// TIA Portal V20 export
DATA_BLOCK "ErrTextList"   // DB371
{ S7_Optimized_Access := 'TRUE' }
// stored: AutoNumber false, MemoryReserve 0
   VAR RETAIN
      language : Array[1..10] of WString[2];   // language for alarm text [ISO639-1]
   END_VAR
   VAR
      writeMessage : Bool;   // write message from program to data block
      err : Array[2000..2205] of Struct   // alarm text
         idProd : UInt;   // producer Id (for Plc: 0=Program_Alarm, 4=SysDiag, 5=MotionControl, 6=Security, 8=GRAPH, 9=ProDiag)
         id : UInt;   // alarm Id
         prio : UInt;   // 0 .. 16 (0-1=info, 2=safety, 3=warning, 4-16=fault)
         alarm : Array[1..8] of WString[150];   // alarm text
      END_STRUCT;
   END_VAR
BEGIN
   language[1] := WSTRING#'de';
   language[2] := WSTRING#'en';
   language[3] := WSTRING#'it';
   language[4] := WSTRING#'fr';
   language[5] := WSTRING#'es';
   err[2031..2040].idProd := 0;
   err[2160..2167].idProd := 0;
   err[2170..2177].idProd := 0;
   err[2180..2187].idProd := 0;
   err[2031..2040].id := 0;
   err[2160..2167].id := 0;
   err[2170..2177].id := 0;
   err[2180..2187].id := 0;
   err[2000..2002].prio := 2;
   err[2004..2005].prio := 2;
   err[2010..2011].prio := 2;
   err[2013..2014].prio := 2;
   err[2016..2017].prio := 2;
   err[2019..2020].prio := 2;
   err[2030..2031].prio := 2;
   err[2032].prio := 0;
   err[2033..2040].prio := 2;
   err[2050].prio := 1;
   err[2052].prio := 0;
   err[2054].prio := 1;
   err[2060].prio := 10;
   err[2075].prio := 2;
   err[2080..2083].prio := 11;
   err[2090..2091].prio := 9;
   err[2100..2102].prio := 10;
   err[2110].prio := 8;
   err[2111].prio := 0;
   err[2120].prio := 12;
   err[2121..2125].prio := 7;
   err[2150].prio := 11;
   err[2151].prio := 10;
   err[2152..2153].prio := 8;
   err[2154].prio := 1;
   err[2156].prio := 1;
   err[2160].prio := 11;
   err[2161].prio := 10;
   err[2162..2163].prio := 8;
   err[2164].prio := 1;
   err[2165].prio := 0;
   err[2166].prio := 1;
   err[2167].prio := 0;
   err[2170].prio := 11;
   err[2171].prio := 10;
   err[2172..2173].prio := 8;
   err[2174].prio := 1;
   err[2175].prio := 0;
   err[2176].prio := 1;
   err[2177].prio := 0;
   err[2180].prio := 11;
   err[2181].prio := 10;
   err[2182..2183].prio := 8;
   err[2184].prio := 1;
   err[2185].prio := 0;
   err[2186].prio := 1;
   err[2187].prio := 0;
   err[2189].prio := 8;
   err[2190].prio := 9;
   err[2000].alarm[1] := WSTRING#'PLC - Not Aus Taster gedrückt am Pc Terminal (-14SB0+HMI.GLD)';
   err[2000].alarm[2] := WSTRING#'PLC - Emergency stop pressed at Pc terminal (-14SB0+HMI.GLD)';
   err[2000].alarm[3] := WSTRING#'PLC - Tasto per arresto di emergenza premuto sul terminale Pc (-14SB0+HMI.GLD)';
   err[2000].alarm[4] := WSTRING#'PLC - Arrêt d`urgence appuyé sur le terminal PC (-14SB0+HMI.GLD)';
   err[2000].alarm[5] := WSTRING#'PLC - Parada de emergencia presionada en terminal Pc (-14SB0+HMI.GLD)';
   err[2001].alarm[1] := WSTRING#'PLC - Not Aus Schlüsselschalter ausgeschalten am Pc Terminal (-14SB1+HMI.GLD)';
   err[2001].alarm[2] := WSTRING#'PLC - Emergency enable key switch off at Pc terminal (-14SB1+HMI.GLD)';
   err[2001].alarm[3] := WSTRING#'PLC - Interruttore a chiave per aresto di emergenza spento sul terminale del PC (-14SB1+HMI.GLD)';
   err[2001].alarm[4] := WSTRING#'PLC - Interrupteur d`urgence désactivé sur le terminal PC (-14SB1+HMI.GLD)';
   err[2001].alarm[5] := WSTRING#'PLC - Interruptor de llave de parada de emergencia apagado en la terminal de la PC (-14SB1+HMI.GLD)';
   err[2002].alarm[1] := WSTRING#'PLC - Quittierung notwendig für Not Aus Taster/Schlüsselschalter am Pc Terminal (-14SB0/1+HMI.GLD)';
   err[2002].alarm[2] := WSTRING#'PLC - Acknowledge required for emergency stop/key switch at Pc terminal (-14SB0/1+HMI.GLD)';
   err[2002].alarm[3] := WSTRING#'PLC - Reset richiesto per pulsante/interrutore di arresto di emergenza sul terminale PC (-14SB0/1+HMI.GLD)';
   err[2002].alarm[4] := WSTRING#'PLC - Reconnaissance nécessaire pour l`arrêt d`urgence/interrupteur à clé sur le terminal PC (-14SB0/1+HMI.GLD)';
   err[2002].alarm[5] := WSTRING#'PLC - Es necesario reiniciar para el botónIinterruptor de emergencia en terminal de PC (-14SB0/1+HMI.GLD)';
   err[2004].alarm[1] := WSTRING#'PLC - Not Aus von externe machine (-XNA+SGV) - aktiv';
   err[2004].alarm[2] := WSTRING#'PLC - Emergency stop from external machine (-XNA+SGV) - active';
   err[2004].alarm[3] := WSTRING#'PLC - Arresto di emergenza da macchina esterna (-XNA+SGV) - attivo';
   err[2004].alarm[4] := WSTRING#'PLC - Arrêt d`urgence depuis une machine externe (-XNA+SGV) - actif';
   err[2004].alarm[5] := WSTRING#'PLC - Parada de emergencia desde máquina externa (-XNA+SGV) - activo';
   err[2005].alarm[1] := WSTRING#'PLC - Not Aus von externe machine (-XNA+SGV) - Quittierung notwendig';
   err[2005].alarm[2] := WSTRING#'PLC - Emergency stop from external machine (-XNA+SGV) - acknowledgement required';
   err[2005].alarm[3] := WSTRING#'PLC - Arresto di emergenza da macchina esterna (-XNA+SGV) - reset necessario';
   err[2005].alarm[4] := WSTRING#'PLC - Arrêt d`urgence depuis une machine externe (-XNA+SGV) - réinitialiser requis';
   err[2005].alarm[5] := WSTRING#'PLC - Parada de emergencia desde máquina externa (-XNA+SGV) - es necesario reiniciar';
   err[2010].alarm[1] := WSTRING#'PLC - Sicherheitsschalter -14SS1.TL+SGV bei Scanner für visuelle Beurteilung oben links - open';
   err[2010].alarm[2] := WSTRING#'PLC - Safety switch -14SS1.TL+SGV at scanner for visual measurement top left - open';
   err[2010].alarm[3] := WSTRING#'PLC - Interruttore di sicurezza -14SS1.TL+SGV sullo scanner per misurazione visiva in alto a sinistra - aperto';
   err[2010].alarm[4] := WSTRING#'PLC - interrupteur de sécurité -14SS1.TL+SGV au scanner pour mesure visuelle en haut à gauche - ouvert';
   err[2010].alarm[5] := WSTRING#'PLC - interruptor de seguridad -14SS1.TL+SGV en el escáner para medición visual arriba a la izquierda - abierto';
   err[2011].alarm[1] := WSTRING#'PLC - Sicherheitsschalter -14SS1.TL+SGV bei Scanner für visuelle Beurteilung oben links - Quittierung notwendig';
   err[2011].alarm[2] := WSTRING#'PLC - safety switch -14SS1.TL+SGV at scanner for visual measurement top left - acknowledge required';
   err[2011].alarm[3] := WSTRING#'PLC - Interruttore di sicurezza -14SS1.TL+SGV sullo scanner per misurazione visiva in alto a sinistra - reset necessario';
   err[2011].alarm[4] := WSTRING#'PLC - interrupteur de sécurité -14SS1.TL+SGV au scanner pour mesure visuelle en haut à gauche - réinitialiser requis';
   err[2011].alarm[5] := WSTRING#'PLC - interruptor de seguridad -14SS1.TL+SGV en el escáner para medición visual arriba a la izquierda - es necesario reiniciar';
   err[2013].alarm[1] := WSTRING#'PLC - Sicherheitsschalter -14SS1.BL+SGV bei Scanner für visuelle Beurteilung unten links - open';
   err[2013].alarm[2] := WSTRING#'PLC - Safety switch -14SS1.BL+SGV at scanner for visual measurement bottom left - open';
   err[2013].alarm[3] := WSTRING#'PLC - Interruttore di sicurezza -14SS1.BL+SGV sullo scanner per misurazione visiva in basso a sinistra - aperto';
   err[2013].alarm[4] := WSTRING#'PLC - interrupteur de sécurité -14SS1.BL+SGV au scanner pour mesure visuelle en bas à gauche - ouvert';
   err[2013].alarm[5] := WSTRING#'PLC - interruptor de seguridad -14SS1.BL+SGV en el escáner para medición visual abajoa la izquierda - abierto';
   err[2014].alarm[1] := WSTRING#'PLC - Sicherheitsschalter -14SS1.BL+SGV bei Scanner für visuelle Beurteilung unten links - Quittierung notwendig';
   err[2014].alarm[2] := WSTRING#'PLC - Safety switch -14SS1.BL+SGV at scanner for visual measurement bottom left - acknowledge required';
   err[2014].alarm[3] := WSTRING#'PLC - Interruttore di sicurezza -14SS1.BL+SGV sullo scanner per misurazione visiva in basso a sinistra - reset necessario';
   err[2014].alarm[4] := WSTRING#'PLC - interrupteur de sécurité -14SS1.BL+SGV au scanner pour mesure visuelle en bas à gauche - réinitialiser requis';
   err[2014].alarm[5] := WSTRING#'PLC - interruptor de seguridad -14SS1.BL+SGV en el escáner para medición visual abajoa la izquierda - es necesario reiniciar';
   err[2016].alarm[1] := WSTRING#'PLC - Sicherheitsschalter -14SS1.TR+SGV bei Scanner für visuelle Beurteilung oben rechts- open';
   err[2016].alarm[2] := WSTRING#'PLC - Safety switch -14SS1.TR+SGV at scanner for visual measurement top right - open';
   err[2016].alarm[3] := WSTRING#'PLC - Interruttore di sicurezza -14SS1.TR+SGV sullo scanner per misurazione visiva in alto a destra - aperto';
   err[2016].alarm[4] := WSTRING#'PLC - interrupteur de sécurité -14SS1.TR+SGV au scanner pour mesure visuelle en haut à droite - ouvert';
   err[2016].alarm[5] := WSTRING#'PLC - interruptor de seguridad -14SS1.TR+SGV en el escáner para medición visual arriba a la derecha - abierto';
   err[2017].alarm[1] := WSTRING#'PLC - Sicherheitsschalter -14SS1.TR+SGV bei Scanner für visuelle Beurteilung oben rechts- Quittierung notwendig';
   err[2017].alarm[2] := WSTRING#'PLC - Safety switch -14SS1.TR+SGV at scanner for visual measurement top right -  acknowledge required';
   err[2017].alarm[3] := WSTRING#'PLC - Interruttore di sicurezza -14SS1.TR+SGV sullo scanner per misurazione visiva in alto a destra - reset necessario';
   err[2017].alarm[4] := WSTRING#'PLC - interrupteur de sécurité -14SS1.TR+SGV au scanner pour mesure visuelle en haut à droite - réinitialiser requis';
   err[2017].alarm[5] := WSTRING#'PLC - interruptor de seguridad -14SS1.TR+SGV en el escáner para medición visual arriba a la derecha - es necesario reiniciar';
   err[2019].alarm[1] := WSTRING#'PLC - Sicherheitsschalter -14SS1.BR+SGV bei Scanner für visuelle Beurteilung unten rechts - open';
   err[2019].alarm[2] := WSTRING#'PLC - Safety switch -14SS1.BR+SGV at scanner for visual measurement bottom right - open';
   err[2019].alarm[3] := WSTRING#'PLC - Interruttore di sicurezza -14SS1.BR+SGV sullo scanner per misurazione visiva in basso a destra - aperto';
   err[2019].alarm[4] := WSTRING#'PLC - interrupteur de sécurité -14SS1.BR+SGV au scanner pour mesure visuelle en bas à droite - ouvert';
   err[2019].alarm[5] := WSTRING#'PLC - interruptor de seguridad -14SS1.BR+SGV en el escáner para medición visual abajo a la derecha - abierto';
   err[2020].alarm[1] := WSTRING#'PLC - Sicherheitsschalter -14SS1.BR+SGV bei Scanner für visuelle Beurteilung unten rechts - Quittierung notwendig';
   err[2020].alarm[2] := WSTRING#'PLC - Safety switch -14SS1.BR+SGV at scanner for visual measurement bottom right -  acknowledge required';
   err[2020].alarm[3] := WSTRING#'PLC - Interruttore di sicurezza -14SS1.BR+SGV sullo scanner per misurazione visiva in basso a destra - reset necessario';
   err[2020].alarm[4] := WSTRING#'PLC - interrupteur de sécurité -14SS1.BR+SGV au scanner pour mesure visuelle en bas à droite - réinitialiser requis';
   err[2020].alarm[5] := WSTRING#'PLC - interruptor de seguridad -14SS1.BR+SGV en el escáner para medición visual abajo a la derecha - es necesario reiniciar';
   err[2030].alarm[1] := WSTRING#'PLC - Sicherheitsschalter -14SS1.TL+SGX bei Scanner für X-Ray oben links - open';
   err[2030].alarm[2] := WSTRING#'PLC - Safety switch -14SS1.TL+SGX at scanner for X-Ray top left - open';
   err[2030].alarm[3] := WSTRING#'PLC - Interruttore di sicurezza -14SS1.TL+SGX sullo scanner per X-Ray in alto a sinistra - aperto';
   err[2030].alarm[4] := WSTRING#'PLC - interrupteur de sécurité -14SS1.TL+SGX au scanner pour X-Ray en haut à gauche - ouvert';
   err[2030].alarm[5] := WSTRING#'PLC - interruptor de seguridad -14SS1.TL+SGX en el escáner para X-Ray arriba a la izquierda - abierto';
   err[2030].alarm[6..8] := WSTRING#'';
   err[2031].alarm[1] := WSTRING#'PLC - Sicherheitsschalter -14SS1.TL+SGX bei Scanner für X-Ray oben links - Quittierung notwendig';
   err[2031].alarm[2] := WSTRING#'PLC - safety switch -14SS1.TL+SGX at scanner for X-Ray top left - acknowledge required';
   err[2031].alarm[3] := WSTRING#'PLC - Interruttore di sicurezza -14SS1.TL+SGX sullo scanner per X-Ray in alto a sinistra - reset necessario';
   err[2031].alarm[4] := WSTRING#'PLC - interrupteur de sécurité -14SS1.TL+SGX au scanner pour X-Ray en haut à gauche - réinitialiser requis';
   err[2031].alarm[5] := WSTRING#'PLC - interruptor de seguridad -14SS1.TL+SGX en el escáner para X-Ray arriba a la izquierda - es necesario reiniciar';
   err[2031].alarm[6..8] := WSTRING#'';
   err[2032].alarm[1..8] := WSTRING#'';
   err[2033].alarm[1] := WSTRING#'PLC - Sicherheitsschalter -14SS1.BL+SGX bei Scanner für X-Ray unten links - open';
   err[2033].alarm[2] := WSTRING#'PLC - Safety switch -14SS1.BL+SGX at scanner for X-Ray bottom left - open';
   err[2033].alarm[3] := WSTRING#'PLC - Interruttore di sicurezza -14SS1.BL+SGX sullo scanner per X-Ray in basso a sinistra - aperto';
   err[2033].alarm[4] := WSTRING#'PLC - interrupteur de sécurité -14SS1.BL+SGX au scanner pour X-Ray en bas à gauche - ouvert';
   err[2033].alarm[5] := WSTRING#'PLC - interruptor de seguridad -14SS1.BL+SGX en el escáner para X-Ray abajoa la izquierda - abierto';
   err[2033].alarm[6..8] := WSTRING#'';
   err[2034].alarm[1] := WSTRING#'PLC - Sicherheitsschalter -14SS1.BL+SGX bei Scanner für X-Ray unten links - Quittierung notwendig';
   err[2034].alarm[2] := WSTRING#'PLC - Safety switch -14SS1.BL+SGX at scanner for X-Rayt bottom left - acknowledge required';
   err[2034].alarm[3] := WSTRING#'PLC - Interruttore di sicurezza -14SS1.BL+SGX sullo scanner per X-Ray in basso a sinistra - reset necessario';
   err[2034].alarm[4] := WSTRING#'PLC - interrupteur de sécurité -14SS1.BL+SGX au scanner pour X-Ray en bas à gauche - réinitialiser requis';
   err[2034].alarm[5] := WSTRING#'PLC - interruptor de seguridad -14SS1.BL+SGX en el escáner para X-Ray abajoa la izquierda - es necesario reiniciar';
   err[2034].alarm[6..8] := WSTRING#'';
   err[2035].alarm[1..8] := WSTRING#'';
   err[2036].alarm[1] := WSTRING#'PLC - Sicherheitsschalter -14SS1.TR+SGX bei Scanner für X-Ray oben rechts- open';
   err[2036].alarm[2] := WSTRING#'PLC - Safety switch -14SS1.TR+SGX at scanner for X-Ray top right - open';
   err[2036].alarm[3] := WSTRING#'PLC - Interruttore di sicurezza -14SS1.TR+SGX sullo scanner per X-Ray in alto a destra - aperto';
   err[2036].alarm[4] := WSTRING#'PLC - interrupteur de sécurité -14SS1.TR+SGX au scanner pour X-Ray en haut à droite - ouvert';
   err[2036].alarm[5] := WSTRING#'PLC - interruptor de seguridad -14SS1.TR+SGX en el escáner para X-Ray arriba a la derecha - abierto';
   err[2036].alarm[6..8] := WSTRING#'';
   err[2037].alarm[1] := WSTRING#'PLC - Sicherheitsschalter -14SS1.TR+SGX bei Scanner für X-Ray oben rechts- Quittierung notwendig';
   err[2037].alarm[2] := WSTRING#'PLC - Safety switch -14SS1.TR+SGX at scanner for X-Ray top right -  acknowledge required';
   err[2037].alarm[3] := WSTRING#'PLC - Interruttore di sicurezza -14SS1.TR+SGX sullo scanner per X-Ray in alto a destra - reset necessario';
   err[2037].alarm[4] := WSTRING#'PLC - interrupteur de sécurité -14SS1.TR+SGX au scanner pour X-Ray en haut à droite - réinitialiser requis';
   err[2037].alarm[5] := WSTRING#'PLC - interruptor de seguridad -14SS1.TR+SGX en el escáner para X-Ray arriba a la derecha - es necesario reiniciar';
   err[2037].alarm[6..8] := WSTRING#'';
   err[2038].alarm[1..8] := WSTRING#'';
   err[2039].alarm[1] := WSTRING#'PLC - Sicherheitsschalter -14SS1.BR+SGX bei Scanner für X-Ray unten rechts - open';
   err[2039].alarm[2] := WSTRING#'PLC - Safety switch -14SS1.BR+SGX at scanner for X-Ray bottom right - open';
   err[2039].alarm[3] := WSTRING#'PLC - Interruttore di sicurezza -14SS1.BR+SGX sullo scanner per X-Ray in basso a destra - aperto';
   err[2039].alarm[4] := WSTRING#'PLC - interrupteur de sécurité -14SS1.BR+SGX au scanner pour X-Ray en bas à droite - ouvert';
   err[2039].alarm[5] := WSTRING#'PLC - interruptor de seguridad -14SS1.BR+SGX en el escáner para X-Ray abajo a la derecha - abierto';
   err[2039].alarm[6..8] := WSTRING#'';
   err[2040].alarm[1] := WSTRING#'PLC - Sicherheitsschalter -14SS1.BR+SGX bei Scanner für X-Ray unten rechts - Quittierung notwendig';
   err[2040].alarm[2] := WSTRING#'PLC - Safety switch -14SS1.BR+SGX at scanner for X-Ray bottom right -  acknowledge required';
   err[2040].alarm[3] := WSTRING#'PLC - Interruttore di sicurezza -14SS1.BR+SGX sullo scanner per X-Ray in basso a destra - reset necessario';
   err[2040].alarm[4] := WSTRING#'PLC - interrupteur de sécurité -14SS1.BR+SGX au scanner pour X-Ray en bas à droite - réinitialiser requis';
   err[2040].alarm[5] := WSTRING#'PLC - interruptor de seguridad -14SS1.BR+SGX en el escáner para X-Ray abajo a la derecha - es necesario reiniciar';
   err[2050].alarm[1] := WSTRING#'PLC - Schlüsselschalter für Einrichtbetrieb am Scanner links aktiviert (-14SB1+SSTL)';
   err[2050].alarm[2] := WSTRING#'PLC - setting mode key switch at scanner left active (-14SB1+SSTL)';
   err[2050].alarm[3] := WSTRING#'PLC - Interruttore a chiave per la modalità di impostazione attivato sullo scanner a sinistra (-14SB1+SSTL)';
   err[2050].alarm[4] := WSTRING#'PLC - commutateur à clé du mode de réglage à gauche du scanner actif (-14SB1+SSTL)';
   err[2050].alarm[5] := WSTRING#'PLC - interruptor de modo de ajuste a la izquierda del escáner activo (-14SB1+SSTL)';
   err[2052].alarm[1] := WSTRING#'PLC - Taster für Freigabe Verstellungen am Scanner links aktiviert (-14SB2+SSTL)';
   err[2052].alarm[2] := WSTRING#'PLC - button to enable adjustments at scanner left active (-14SB21+SSTL)';
   err[2052].alarm[3] := WSTRING#'PLC - pulsante per abilitare le assi attivato sullo scanner a sinistra (-14SB2+SSTL)';
   err[2052].alarm[4] := WSTRING#'PLC - bouton pour activer les réglages à gauche du scanner actif (-14SB2+SSTL)';
   err[2052].alarm[5] := WSTRING#'PLC - botón para habilitar ajustes a la izquierda del escáner activo (-14SB2+SSTL)';
   err[2054].alarm[1] := WSTRING#'PLC - Kühlgeräte wurden am Scanner rechts deaktiviert (-14SB2+SSTL)';
   err[2054].alarm[2] := WSTRING#'PLC - air-conditioning is switched off at scanner right (-0SH1+SSTR)';
   err[2054].alarm[3] := WSTRING#'PLC - l`aria condizionata è stata spenta sullo scanner a destra (-14SB2+SSTL)';
   err[2054].alarm[4] := WSTRING#'PLC - la climatisation est éteinte au niveau du scanner à droite (-14SB2+SSTL)';
   err[2054].alarm[5] := WSTRING#'PLC - El aire acondicionado está apagado en el escáner a la derecha (-14SB2+SSTL)';
   err[2060].alarm[1] := WSTRING#'PLC - Störung Sicherheitsmodule';
   err[2060].alarm[2] := WSTRING#'PLC - fault safety modules plc';
   err[2060].alarm[3] := WSTRING#'PLC - errore sui moduli di sicurezza';
   err[2060].alarm[4] := WSTRING#'PLC - modules de sécurité contre les défauts';
   err[2060].alarm[5] := WSTRING#'PLC - módulos de seguridad contra fallas';
   err[2075].alarm[1] := WSTRING#'PLC - Sicherheitsbereich Extern oder Intern ausgeschalten - Quittierung notwendig';
   err[2075].alarm[2] := WSTRING#'PLC - safety area internal/external switched off - acknowledge required';
   err[2075].alarm[3] := WSTRING#'PLC - area di sicurezza interna/esterna spenta- reset necessario';
   err[2075].alarm[4] := WSTRING#'PLC - zone de sécurité interne/externe désactivée - réinitialiser requis';
   err[2075].alarm[5] := WSTRING#'PLC - area de seguridad interna/externa apagada - es necesario reiniciar';
   err[2080].alarm[1] := WSTRING#'PLC - Störung Rückführung Sicherheitsbereich - Bereich laser (-14KA1+SGV)';
   err[2080].alarm[2] := WSTRING#'PLC - fault safety feedback monitoring - area laser (-14KA1+SGV)';
   err[2080].alarm[3] := WSTRING#'PLC - errore monitoraggio feedback di sicurezza - area laser (-14KA1+SGV)';
   err[2080].alarm[4] := WSTRING#'PLC - défaut surveillance de la sécurité - zone laser (-14KA1+SGV)';
   err[2080].alarm[5] := WSTRING#'PLC - fallo de monitoreo de retroalimentación de seguridad - área de láser (-14KA1+SGV)';
   err[2081].alarm[1] := WSTRING#'PLC - Störung Rückführung Sicherheitsbereich - Bereich Verstellung (-14KA2+SGV)';
   err[2081].alarm[2] := WSTRING#'PLC - fault safety feedback monitoring - area adjustment (-14KA2+SGV)';
   err[2081].alarm[3] := WSTRING#'PLC - errore monitoraggio feedback di sicurezza - area posizionamento (-14KA2+SGV)';
   err[2081].alarm[4] := WSTRING#'PLC - défaut surveillance de la sécurité - zone réglage (-14KA2+SGV)';
   err[2081].alarm[5] := WSTRING#'PLC - fallo de monitoreo de retroalimentación de seguridad - área de ajuste (-14KA2+SGV)';
   err[2082].alarm[1] := WSTRING#'PLC - Störung Rückführung Sicherheitsbereich - Bereich Verstellung LINMOT (8U1+SGV)';
   err[2082].alarm[2] := WSTRING#'PLC - fault safety feedback monitoring - area adjustment LINMOT (8U1+SGV)';
   err[2082].alarm[3] := WSTRING#'PLC - errore monitoraggio feedback di sicurezza - area posizionamento LINMOT (8U1+SGV)';
   err[2082].alarm[4] := WSTRING#'PLC - défaut surveillance de la sécurité - zone réglage LINMOT (8U1+SGV)';
   err[2082].alarm[5] := WSTRING#'PLC - fallo de monitoreo de retroalimentación de seguridad - área de ajuste LINMOT (8U1+SGV)';
   err[2083].alarm[1] := WSTRING#'PLC - Störung Rückführung Sicherheitsbereich - Bereich X-Ray (-5AX1+SGX)';
   err[2083].alarm[2] := WSTRING#'PLC - fault safety feedback monitoring - area X-Ray (-5AX1+SGX)';
   err[2083].alarm[3] := WSTRING#'PLC - errore monitoraggio feedback di sicurezza - area X-Ray (-5AX1+SGX)';
   err[2083].alarm[4] := WSTRING#'PLC - défaut surveillance de la sécurité - zone X-Ray (-5AX1+SGX)';
   err[2083].alarm[5] := WSTRING#'PLC - fallo de monitoreo de retroalimentación de seguridad - área X-Ray (-5AX1+SGX)';
   err[2090].alarm[1] := WSTRING#'PLC - Störung Lichtschranke im Scanner für visuelle Beurteilung (-1BTR2+SGV)';
   err[2090].alarm[2] := WSTRING#'PLC - fault light barrier in scanner for visual measurement (-1BTR2+SGV)';
   err[2090].alarm[3] := WSTRING#'PLC - errore sensore nel scanner per misurazione visiva (-1BTR2+SGV)';
   err[2090].alarm[4] := WSTRING#'PLC - défaut capteur dans le scanner pour la mesure visuelle (-1BTR2+SGV)';
   err[2090].alarm[5] := WSTRING#'PLC - fallo de sensor en escáner para medición visual (-1BTR2+SGV)';
   err[2091].alarm[1] := WSTRING#'PLC - Störung Lichtschranke vor Scanner für X-Ray (-1BTR2+SGX)';
   err[2091].alarm[2] := WSTRING#'PLC - fault light barrier before scanner for X-Ray (-1BTR2+SGX)';
   err[2091].alarm[3] := WSTRING#'PLC - errore sensore prime dello scanner per X-Ray (-1BTR2+SGX)';
   err[2091].alarm[4] := WSTRING#'PLC - défaut capteur avant le scanner pour X-Ray (-1BTR2+SGX)';
   err[2091].alarm[5] := WSTRING#'PLC - fallo de sensor antes escáner para X-Ray (-1BTR2+SGX)';
   err[2100].alarm[1] := WSTRING#'PLC - Störung Encoder vor Scanner (-1BCI1+GLD)';
   err[2100].alarm[2] := WSTRING#'PLC - fault encoder before scanner (-1BCI1+GLD)';
   err[2100].alarm[3] := WSTRING#'PLC - errore encoder davanti allo scanner (-1BCI1+GLD)';
   err[2100].alarm[4] := WSTRING#'PLC - défaut codeur avant le scanner (-1BCI1+GLD)';
   err[2100].alarm[5] := WSTRING#'PLC - fallo de codificador antes escáner (-1BCI1+GLD)';
   err[2101].alarm[1] := WSTRING#'PLC - Störung Encoder im Scanner (-1BCM1+GLD)';
   err[2101].alarm[2] := WSTRING#'PLC - fault encoder in scanner (-1BCM1+GLD)';
   err[2101].alarm[3] := WSTRING#'PLC - errore encoder nello scanner (-1BCM1+GLD)';
   err[2101].alarm[4] := WSTRING#'PLC - défaut codeur dans le scanner (-1BCM1+GLD)';
   err[2101].alarm[5] := WSTRING#'PLC - fallo de codificador en escáner (-1BCM1+GLD)';
   err[2102].alarm[1] := WSTRING#'PLC - Störung Encoder nach Scanner (-1BCO1+GLD)';
   err[2102].alarm[2] := WSTRING#'PLC - fault encoder after scanner (-1BCO1+GLD)';
   err[2102].alarm[3] := WSTRING#'PLC - errore encoder dopo lo scanner (-1BCO1+GLD)';
   err[2102].alarm[4] := WSTRING#'PLC - défaut codeur après le scanner (-1BCO1+GLD)';
   err[2102].alarm[5] := WSTRING#'PLC - fallo de codificador después del escáner (-1BCO1+GLD)';
   err[2110].alarm[1] := WSTRING#'PLC - Störung Kommunikation mit Goldeneye Pc';
   err[2110].alarm[2] := WSTRING#'PLC - fault communication with Goldeneye Pc';
   err[2110].alarm[3] := WSTRING#'PLC - errore comunicazione con Goldeneye Pc';
   err[2110].alarm[4] := WSTRING#'PLC - défaut communication avec Goldeneye Pc';
   err[2110].alarm[5] := WSTRING#'PLC - fallo comunicación con Goldeneye Pc';
   err[2111].alarm[1] := WSTRING#'PLC - Keine Freigabe vom Goldeneye Pc für den Einzug';
   err[2111].alarm[2] := WSTRING#'PLC - no release from Goldeneye Pc to infeed';
   err[2111].alarm[3] := WSTRING#'PLC - nessun permesso dal Goldeneye Pc per alimentazione ';
   err[2111].alarm[4] := WSTRING#'PLC - pas de sortie de Goldeneye PC pour infeed';
   err[2111].alarm[5] := WSTRING#'PLC - no hay liberación de Goldeneye Pc para la entrada';
   err[2120].alarm[1] := WSTRING#'PLC - Störung elektronischer Schutzschalter (-0F1.1+SGV)';
   err[2120].alarm[2] := WSTRING#'PLC - fault electronic circuit breaker (-0F1.1+SGV)';
   err[2120].alarm[3] := WSTRING#'PLC - errore interruttore elettronico (-0F1.1+SGV)';
   err[2120].alarm[4] := WSTRING#'PLC - défaut disjoncteur électronique (-0F1.1+SGV)';
   err[2120].alarm[5] := WSTRING#'PLC - fallo disyuntor electrónico (-0F1.1+SGV)';
   err[2121].alarm[1] := WSTRING#'PLC - Störung Kühlgerät 1 bei Scanner für visuelle Beurteilung (-0E1+SGV)';
   err[2121].alarm[2] := WSTRING#'PLC - fault air-conditioning unit 1 for scannerhousing visual measurement (-0E1+SGV)';
   err[2121].alarm[3] := WSTRING#'PLC - errore unità di raffreddamento 1 per scanner per misurazione visiva (-0E1+SGV)';
   err[2121].alarm[4] := WSTRING#'PLC - défaut unité de refroidissement 1 chez scanner pour mesure visuelle (-0E1+SGV)';
   err[2121].alarm[5] := WSTRING#'PLC - fallo unidad de refrigeración 1 para escáner para medición visual (-0E1+SGV)';
   err[2122].alarm[1] := WSTRING#'PLC - Störung Kühlgerät bei Scanner für X-Ray (-0E2+SGX)';
   err[2122].alarm[2] := WSTRING#'PLC - fault air-conditioning unit for scannerhousing  X-Ray (-0E2+SGX)';
   err[2122].alarm[3] := WSTRING#'PLC - errore unità di raffreddamento per scanner per X-Ray (-0E2+SGX)';
   err[2122].alarm[4] := WSTRING#'PLC - défaut unité de refroidissement chez scanner pour X-Ray (-0E2+SGX)';
   err[2122].alarm[5] := WSTRING#'PLC - fallo unidad de refrigeración para escáner para X-Ray (-0E2+SGX)';
   err[2123].alarm[1] := WSTRING#'PLC - Störung Kühlgerät 2 bei Scanner für visuelle Beurteilung (-0E1.1+SGV)';
   err[2123].alarm[2] := WSTRING#'PLC - fault air-conditioning unit 2 for scannerhousing visual measurement (-0E1.1+SGV)';
   err[2123].alarm[3] := WSTRING#'PLC - errore unità di raffreddamento 2 per scanner per misurazione visiva (-0E1.1+SGV)';
   err[2123].alarm[4] := WSTRING#'PLC - défaut unité de refroidissement 2 chez scanner pour mesure visuelle (-0E1.1+SGV)';
   err[2123].alarm[5] := WSTRING#'PLC - fallo unidad de refrigeración 2 para escáner para medición visual (-0E1.1+SGV)';
   err[2124].alarm[1] := WSTRING#'PLC - Störung Entfeuchter bei Scanner für (-0E1.2+SGV)';
   err[2124].alarm[2] := WSTRING#'PLC - fault dehumidifier for scannerhousing (-0E1.2+SGV)';
   err[2124].alarm[3] := WSTRING#'PLC - errore deumidificatore per scanner (-0E1.2+SGV)';
   err[2124].alarm[4] := WSTRING#'PLC - défaut déshumidificateur chez scanner (-0E1.2+SGV)';
   err[2124].alarm[5] := WSTRING#'PLC - fallo deshumidificador para escáner (-0E1.2+SGV)';
   err[2125].alarm[1] := WSTRING#'PLC - Störung Kommunikationsschnittstelle zwischen Pc und Sps ist unterschiedlich';
   err[2125].alarm[2] := WSTRING#'PLC - fault communication interface between Pc and Plc is different';
   err[2125].alarm[3] := WSTRING#'PLC - errore l`interfaccia di comunicazione tra Pc e Plc è diversa';
   err[2125].alarm[4] := WSTRING#'PLC - défaut l`interface de communication entre le PC et Plc est différente';
   err[2125].alarm[5] := WSTRING#'PLC - fallo La interfaz de comunicación entre PC y PLC es diferente';
   err[2140].alarm[1] := WSTRING#'PLC - Verstellung Scanner wurde temporär deaktiviert, kann nur mehr manuel verfahren werden (-8M1.B+SGV)';
   err[2140].alarm[2] := WSTRING#'PLC - adjustment scannerhousing is deactivated temporaly, you can move only manualy (-8M1.B+SGV)';
   err[2140].alarm[3] := WSTRING#'PLC - posizionamento scanner è temporaneamente disattivato, è possibile muoverlo solo manualmente (-8M1.B+SGV)';
   err[2140].alarm[4] := WSTRING#'PLC - positionnement de scanner est temporairement désactivé, vous ne pouvez le déplacer que manuellement (-8M1.B+SGV)';
   err[2140].alarm[5] := WSTRING#'PLC - el ajuste de del escáner se desactiva temporalmente, solo se puede mover manualmente (-8M1.B+SGV)';
   err[2141].alarm[1] := WSTRING#'PLC - Verstellung Messbalken oben wurde temporär deaktiviert, kann nur mehr manuel verfahren werden (-8M1.T+SGV)';
   err[2141].alarm[2] := WSTRING#'PLC - adjustment metering bar top is deactivated temporaly, you can move only manualy (-8M1.T+SGV)';
   err[2141].alarm[3] := WSTRING#'PLC - posizionamento barra di misura superiore è temporaneamente disattivato, è possibile muoverlo solo manualmente (-8M1.T+SGV)';
   err[2141].alarm[4] := WSTRING#'PLC - positionnement de barre de mesure supérieure est temporairement désactivé, vous ne pouvez le déplacer que manuellement (-8M1.T+SGV)';
   err[2141].alarm[5] := WSTRING#'PLC - el ajuste de barra de medición superior se desactiva temporalmente, solo se puede mover manualmente (-8M1.T+SGV)';
   err[2142].alarm[1] := WSTRING#'PLC - Verstellung Messbalken links wurde temporär deaktiviert, kann nur mehr manuel verfahren werden (-8M1.L+SGV)';
   err[2142].alarm[2] := WSTRING#'PLC - adjustment metering bar left is deactivated temporaly, you can move only manualy (-8M1.L+SGV)';
   err[2142].alarm[3] := WSTRING#'PLC - posizionamento barra di misura di sinistra è temporaneamente disattivato, è possibile muoverlo solo manualmente (-8M1.L+SGV)';
   err[2142].alarm[4] := WSTRING#'PLC - positionnement de barre de mesure gauche est temporairement désactivé, vous ne pouvez le déplacer que manuellement (-8M1L+SGV)';
   err[2142].alarm[5] := WSTRING#'PLC - el ajuste de barra de medición izquierda se desactiva temporalmente, solo se puede mover manualmente (-8M1.L+SGV)';
   err[2143].alarm[1] := WSTRING#'PLC - Verstellung Messbalken rechts wurde temporär deaktiviert, kann nur mehr manuel verfahren werden (-8M1.R+SGV)';
   err[2143].alarm[2] := WSTRING#'PLC - adjustment metering bar right is deactivated temporaly, you can move only manualy (-8M1.R+SGV)';
   err[2143].alarm[3] := WSTRING#'PLC - posizionamento barra di misura di destra è temporaneamente disattivato, è possibile muoverlo solo manualmente (-8M1.R+SGV)';
   err[2143].alarm[4] := WSTRING#'PLC - positionnement de barre de mesure à droite est temporairement désactivé, vous ne pouvez le déplacer que manuellement (-8M1.R+SGV)';
   err[2143].alarm[5] := WSTRING#'PLC - el ajuste de barra de medición derecha se desactiva temporalmente, solo se puede mover manualmente (-8M1.R+SGV)';
   err[2144].alarm[1] := WSTRING#'PLC - Kühlgerät 1 bei Scanner für visuelle Beurteilung wurde temporär deaktiviert (-0E1+SGV)';
   err[2144].alarm[2] := WSTRING#'PLC - air-conditioning unit 1 for scannerhousing visual measurement is deactivated temporaly (-0E1+SGV)';
   err[2144].alarm[3] := WSTRING#'PLC - unità di raffreddamento 1 per scanner per misurazione visiva è temporaneamente disattivato (-0E1+SGV)';
   err[2144].alarm[4] := WSTRING#'PLC - unité de refroidissement 1 chez scanner pour mesure visuelle est temporairement désactivé (-0E1+SGV)';
   err[2144].alarm[5] := WSTRING#'PLC - unidad de refrigeración 1 para escáner para medición visual se desactiva temporalmente (-0E1+SGV)';
   err[2145].alarm[1] := WSTRING#'PLC - Kühlgerät 2 bei Scanner für visuelle Beurteilung wurde temporär deaktiviert (-0E1.1+SGV)';
   err[2145].alarm[2] := WSTRING#'PLC - air-conditioning unit 2 for scannerhousing visual measurement is deactivated temporaly (-0E1.1+SGV)';
   err[2145].alarm[3] := WSTRING#'PLC - unità di raffreddamento 2 per scanner per misurazione visiva è temporaneamente disattivato (-0E1.1+SGV)';
   err[2145].alarm[4] := WSTRING#'PLC - unité de refroidissement 2 chez scanner pour mesure visuelle est temporairement désactivé (-0E1.1+SGV)';
   err[2145].alarm[5] := WSTRING#'PLC - unidad de refrigeración 2 para escáner para medición visual se desactiva temporalmente (-0E1.1+SGV)';
   err[2146].alarm[1] := WSTRING#'PLC - Kühlgerät bei Scanner für X-Ray wurde temporär deaktiviert (-0E2+SGX)';
   err[2146].alarm[2] := WSTRING#'PLC - air-conditioning unit for scannerhousing X-Ray measurement is deactivated temporaly (-0E2+SGX)';
   err[2146].alarm[3] := WSTRING#'PLC - unità di raffreddamento per scanner per X-Ray è temporaneamente disattivato (-0E2+SGX)';
   err[2146].alarm[4] := WSTRING#'PLC - unité de refroidissement chez scanner pour X-Ray est temporairement désactivé (-0E2+SGX)';
   err[2146].alarm[5] := WSTRING#'PLC - unidad de refrigeración 1 para escáner paraX-Ray se desactiva temporalmente (-0E2+SGX)';
   err[2147].alarm[1] := WSTRING#'PLC - Entfeuchter bei Scanner wurde temporär deaktiviert (-0E3+SGX)';
   err[2147].alarm[2] := WSTRING#'PLC - dehumidifier for scannerhousing is deactivated temporaly (-0E3+SGX)';
   err[2147].alarm[3] := WSTRING#'PLC - deumidificatore per scanner è temporaneamente disattivato (-0E3+SGX)';
   err[2147].alarm[4] := WSTRING#'PLC - déshumidificateur chez scanner est temporairement désactivé (-0E3+SGX)';
   err[2147].alarm[5] := WSTRING#'PLC - deshumidificador para escáner se desactiva temporalmente (-0E3+SGX)';
   err[2150].alarm[1] := WSTRING#'PLC - Störung Verstellung Scanner (-8M1.B+SGV)';
   err[2150].alarm[2] := WSTRING#'PLC - fault adjustment scannerhousing (-8M1.B+SGV)';
   err[2150].alarm[3] := WSTRING#'PLC - errore posizionamento scanner (-8M1.B+SGV)';
   err[2150].alarm[4] := WSTRING#'PLC - défaut positionnement de scanner (-8M1.B+SGV)';
   err[2150].alarm[5] := WSTRING#'PLC - fallo el ajuste de del escáner (-8M1.B+SGV)';
   err[2151].alarm[1] := WSTRING#'PLC - Störung Encoder - Verstellung Scanner (-8B1.B+SGV)';
   err[2151].alarm[2] := WSTRING#'PLC - fault encoder - adjustment scannerhousing (-8B1.B+SGV)';
   err[2151].alarm[3] := WSTRING#'PLC - errore encoder - posizionamento scanner (-8B1.B+SGV)';
   err[2151].alarm[4] := WSTRING#'PLC - défaut codeur - positionnement de scanner (-8B1.B+SGV)';
   err[2151].alarm[5] := WSTRING#'PLC - fallo codificador - el ajuste de del escáner (-8B1.B+SGV)';
   err[2152].alarm[1] := WSTRING#'PLC - Störung Sensor Endstellung links - Verstellung Scanner (-8S1.B+SGV)';
   err[2152].alarm[2] := WSTRING#'PLC - fault sensor limit switch position left - adjustment scannerhousing (-8S1.B+SGV)';
   err[2152].alarm[3] := WSTRING#'PLC - errore sensore posizione sinistra - posizionamento scanner (-8S1.B+SGV)';
   err[2152].alarm[4] := WSTRING#'PLC - défaut capteur position du fin de course à gauche - positionnement de scanner (-8S1.B+SGV)';
   err[2152].alarm[5] := WSTRING#'PLC - fallo sensor posición de límite a la izquierda - el ajuste de del escáner (-8S1.B+SGV)';
   err[2153].alarm[1] := WSTRING#'PLC - Störung Sensor Endstellung rechts - Verstellung Scanner (-8S2.B+SGV)';
   err[2153].alarm[2] := WSTRING#'PLC - fault sensor limit switch position right - adjustment scannerhousing (-8S2.B+SGV)';
   err[2153].alarm[3] := WSTRING#'PLC - errore sensore posizione destra - posizionamento scanner (-8S2.B+SGV)';
   err[2153].alarm[4] := WSTRING#'PLC - défaut capteur position du fin de course à droite - positionnement de scanner (-8S2.B+SGV)';
   err[2153].alarm[5] := WSTRING#'PLC - fallo sensor posición de límite a la derecha - el ajuste de del escáner (-8S2.B+SGV)';
   err[2154].alarm[1] := WSTRING#'PLC - Verstellung Scanner nicht referenziert, händisch neu referenzieren (-8M1.B+SGV)';
   err[2154].alarm[2] := WSTRING#'PLC - adjustment scannerhousing reference not ok, reference manualy (-8M1.B+SGV)';
   err[2154].alarm[3] := WSTRING#'PLC - posizionamento scanner riferimento non coretto, fare corsa di riferimento (-8M1.B+SGV)';
   err[2154].alarm[4] := WSTRING#'PLC - positionnement de scanner référence non correcte, manuel de référence (-8M1.B+SGV)';
   err[2154].alarm[5] := WSTRING#'PLC - el ajuste de del escáner referencia no ok, manual de referencia (-8M1.B+SGV)';
   err[2155].alarm[1] := WSTRING#'PLC - Verstellung Scanner Referenzfahrt aktiv  (-8M1.B+SGV)';
   err[2155].alarm[2] := WSTRING#'PLC - adjustment scannerhousing reference run active (-8M1.B+SGV)';
   err[2155].alarm[3] := WSTRING#'PLC - posizionamento scanner corsa di riferimento attiva (-8M1.B+SGV)';
   err[2155].alarm[4] := WSTRING#'PLC - positionnement de scanner exécution de référence active (-8M1.B+SGV)';
   err[2155].alarm[5] := WSTRING#'PLC - el ajuste de del escáner ejecución de referencia activa (-8M1.B+SGV)';
   err[2156].alarm[1] := WSTRING#'PLC - Verstellung Scanner nicht in Position (-8M1.B+SGV)';
   err[2156].alarm[2] := WSTRING#'PLC - adjustment scannerhousing not in position (-8M1.B+SGV)';
   err[2156].alarm[3] := WSTRING#'PLC - posizionamento scanner non in posizione (-8M1.B+SGV)';
   err[2156].alarm[4] := WSTRING#'PLC - positionnement de scanner pas en position (-8M1.B+SGV)';
   err[2156].alarm[5] := WSTRING#'PLC - el ajuste de del escáner no está en posición (-8M1.B+SGV)';
   err[2157].alarm[1] := WSTRING#'PLC - Verstellung Scanner am Pc auf Hand geschalten (-8M1.B+SGV)';
   err[2157].alarm[2] := WSTRING#'PLC - adjustment scannerhousing set on manual mode on Pc (-8M1.B+SGV)';
   err[2157].alarm[3] := WSTRING#'PLC - posizionamento scanner attivata modalità manuale sul Pc (-8M1.B+SGV)';
   err[2157].alarm[4] := WSTRING#'PLC - positionnement de scanner passé en mode manuel sur le Pc (-8M1.B+SGV)';
   err[2157].alarm[5] := WSTRING#'PLC - el ajuste de del escáner cambiado a manual en la Pc (-8M1.B+SGV)';
   err[2160].alarm[1] := WSTRING#'PLC - Störung Verstellung Messbalken oben (-8M1.T+SGV)';
   err[2160].alarm[2] := WSTRING#'PLC - fault adjustment metering bar top (-8M1.T+SGV)';
   err[2160].alarm[3] := WSTRING#'PLC - errore posizionamento barra di misura superiore (-8M1.T+SGV)';
   err[2160].alarm[4] := WSTRING#'PLC - défaut positionnement de barre de mesure supérieure (-8M1.T+SGV)';
   err[2160].alarm[5] := WSTRING#'PLC - fallo el ajuste de barra de medición superior (-8M1.T+SGV)';
   err[2160].alarm[6..8] := WSTRING#'';
   err[2161].alarm[1] := WSTRING#'PLC - Störung Encoder - Verstellung Messbalken oben (-8B1.T+SGV)';
   err[2161].alarm[2] := WSTRING#'PLC - fault encoder - adjustment metering bar top (-8B1.T+SGV)';
   err[2161].alarm[3] := WSTRING#'PLC - errore encoder - posizionamento barra di misura superiore (-8B1.T+SGV)';
   err[2161].alarm[4] := WSTRING#'PLC - défaut codeur - positionnement de barre de mesure supérieure (-8B1.T+SGV)';
   err[2161].alarm[5] := WSTRING#'PLC - fallo codificador - el ajuste de barra de medición superior (-8B1.T+SGV)';
   err[2161].alarm[6..8] := WSTRING#'';
   err[2162].alarm[1] := WSTRING#'PLC - Störung Sensor Endstellung links - Verstellung Messbalken oben (-8S1.T+SGV)';
   err[2162].alarm[2] := WSTRING#'PLC - fault sensor limit switch position left - adjustment metering bar top (-8S1.T+SGV)';
   err[2162].alarm[3] := WSTRING#'PLC - errore sensore posizione sinistra - posizionamento barra di misura superiore (-8S1.T+SGV)';
   err[2162].alarm[4] := WSTRING#'PLC - défaut capteur position du fin de course à gauche - positionnement de barre de mesure supérieure (-8S1.T+SGV)';
   err[2162].alarm[5] := WSTRING#'PLC - fallo sensor posición de límite a la izquierda - el ajuste de barra de medición superior (-8S1.T+SGV)';
   err[2162].alarm[6..8] := WSTRING#'';
   err[2163].alarm[1] := WSTRING#'PLC - Störung Sensor Endstellung rechts - Verstellung Messbalken oben (-8S2.T+SGV)';
   err[2163].alarm[2] := WSTRING#'PLC - fault sensor limit switch position right - adjustment metering bar top (-8S2.T+SGV)';
   err[2163].alarm[3] := WSTRING#'PLC - errore sensore posizione destra - posizionamento barra di misura superiore (-8S2.T+SGV)';
   err[2163].alarm[4] := WSTRING#'PLC - défaut capteur position du fin de course à droite - positionnement de barre de mesure supérieure (-8S2.T+SGV)';
   err[2163].alarm[5] := WSTRING#'PLC - fallo sensor posición de límite a la derecha - el ajuste de barra de medición superior (-8S2.T+SGV)';
   err[2163].alarm[6..8] := WSTRING#'';
   err[2164].alarm[1] := WSTRING#'PLC - Verstellung Messbalken oben nicht referenziert, händisch neu referenzieren (-8M1.T+SGV)';
   err[2164].alarm[2] := WSTRING#'PLC - adjustment metering bar top reference not ok, reference manualy (-8M1.T+SGV)';
   err[2164].alarm[3] := WSTRING#'PLC - posizionamento barra di misura superiore riferimento non coretto, fare corsa di riferimento (-8M1.T+SGV)';
   err[2164].alarm[4] := WSTRING#'PLC - positionnement de barre de mesure supérieure référence non correcte, manuel de référence (-8M1.T+SGV)';
   err[2164].alarm[5] := WSTRING#'PLC - el ajuste de barra de medición superior referencia no ok, manual de referencia (-8M1.T+SGV)';
   err[2164].alarm[6..8] := WSTRING#'';
   err[2165].alarm[1] := WSTRING#'PLC - Verstellung Messbalken oben Referenzfahrt aktiv  (-8M1.T+SGV)';
   err[2165].alarm[2] := WSTRING#'PLC - adjustment metering bar top reference run active (-8M1.T+SGV)';
   err[2165].alarm[3] := WSTRING#'PLC - posizionamento barra di misura superiore corsa di riferimento attiva (-8M1.T+SGV)';
   err[2165].alarm[4] := WSTRING#'PLC - positionnement de barre de mesure supérieure exécution de référence active (-8M1.T+SGV)';
   err[2165].alarm[5] := WSTRING#'PLC - el ajuste de barra de medición superior ejecución de referencia activa (-8M1.T+SGV)';
   err[2165].alarm[6..8] := WSTRING#'';
   err[2166].alarm[1] := WSTRING#'PLC - Verstellung Messbalken oben nicht in Position (-8M1.T+SGV)';
   err[2166].alarm[2] := WSTRING#'PLC - adjustment metering bar top not in position (-8M1.T+SGV)';
   err[2166].alarm[3] := WSTRING#'PLC - posizionamento barra di misura superiore non in posizione (-8M1.T+SGV)';
   err[2166].alarm[4] := WSTRING#'PLC - positionnement de barre de mesure supérieure pas en position (-8M1.T+SGV)';
   err[2166].alarm[5] := WSTRING#'PLC - el ajuste de barra de medición superior no está en posición (-8M1.T+SGV)';
   err[2166].alarm[6..8] := WSTRING#'';
   err[2167].alarm[1] := WSTRING#'PLC - Verstellung Messbalken oben am Pc auf Hand geschalten (-8M1.T+SGV)';
   err[2167].alarm[2] := WSTRING#'PLC - adjustment metering bar top set on manual mode on Pc (-8M1.T+SGV)';
   err[2167].alarm[3] := WSTRING#'PLC - posizionamento barra di misura superiore attivata modalità manuale sul Pc (-8M1.T+SGV)';
   err[2167].alarm[4] := WSTRING#'PLC - positionnement de barre de mesure supérieure passé en mode manuel sur le Pc (-8M1.T+SGV)';
   err[2167].alarm[5] := WSTRING#'PLC - el ajuste de barra de medición superior cambiado a manual en la Pc (-8M1.T+SGV)';
   err[2170].alarm[1] := WSTRING#'PLC - Störung Verstellung Messbalken links (-8M1.L+SGV)';
   err[2170].alarm[2] := WSTRING#'PLC - fault adjustment metering bar left (-8M1.L+SGV)';
   err[2170].alarm[3] := WSTRING#'PLC - errore posizionamento barra di misura di sinistra (-8M1.L+SGV)';
   err[2170].alarm[4] := WSTRING#'PLC - défaut positionnement de barre de mesure gauche (-8M1.L+SGV)';
   err[2170].alarm[5] := WSTRING#'PLC - fallo el ajuste de barra de medición izquierda (-8M1.L+SGV)';
   err[2170].alarm[6..8] := WSTRING#'';
   err[2171].alarm[1] := WSTRING#'PLC - Störung Encoder - Verstellung Messbalken links (-8B1.L+SGV)';
   err[2171].alarm[2] := WSTRING#'PLC - fault encoder - adjustment metering bar left (-8B1.L+SGV)';
   err[2171].alarm[3] := WSTRING#'PLC - errore encoder - posizionamento barra di misura di sinistra (-8B1.L+SGV)';
   err[2171].alarm[4] := WSTRING#'PLC - défaut codeur - positionnement de barre de mesure gauche (-8B1.L+SGV)';
   err[2171].alarm[5] := WSTRING#'PLC - fallo codificador - el ajuste de barra de medición izquierda (-8B1.L+SGV)';
   err[2171].alarm[6..8] := WSTRING#'';
   err[2172].alarm[1] := WSTRING#'PLC - Störung Sensor Endstellung links - Verstellung Messbalken links (-8S1.L+SGV)';
   err[2172].alarm[2] := WSTRING#'PLC - fault sensor limit switch position left - adjustment metering bar left (-8S1.L+SGV)';
   err[2172].alarm[3] := WSTRING#'PLC - errore sensore posizione sinistra - posizionamento barra di misura di sinistra (-8S1.L+SGV)';
   err[2172].alarm[4] := WSTRING#'PLC - défaut capteur position du fin de course à gauche - positionnement de barre de mesure gauche (-8S1.L+SGV)';
   err[2172].alarm[5] := WSTRING#'PLC - fallo sensor posición de límite a la izquierda - el ajuste de barra de medición izquierda (-8S1.L+SGV)';
   err[2172].alarm[6..8] := WSTRING#'';
   err[2173].alarm[1] := WSTRING#'PLC - Störung Sensor Endstellung rechts - Verstellung Messbalken links (-8S2.L+SGV)';
   err[2173].alarm[2] := WSTRING#'PLC - fault sensor limit switch position right - adjustment metering bar left (-8S2.L+SGV)';
   err[2173].alarm[3] := WSTRING#'PLC - errore sensore posizione destra - posizionamento barra di misura di sinistra (-8S2.L+SGV)';
   err[2173].alarm[4] := WSTRING#'PLC - défaut capteur position du fin de course à droite - positionnement de barre de mesure gauche (-8S2.L+SGV)';
   err[2173].alarm[5] := WSTRING#'PLC - fallo sensor posición de límite a la derecha - el ajuste de barra de medición izquierda (-8S2.L+SGV)';
   err[2173].alarm[6..8] := WSTRING#'';
   err[2174].alarm[1] := WSTRING#'PLC - Verstellung Messbalken links nicht referenziert, händisch neu referenzieren (-8M1.L+SGV)';
   err[2174].alarm[2] := WSTRING#'PLC - adjustment metering bar left reference not ok, reference manualy (-8M1.L+SGV)';
   err[2174].alarm[3] := WSTRING#'PLC - posizionamento barra di misura di sinistra riferimento non coretto, fare corsa di riferimento (-8M1.L+SGV)';
   err[2174].alarm[4] := WSTRING#'PLC - positionnement de barre de mesure gauche référence non correcte, manuel de référence (-8M1.L+SGV)';
   err[2174].alarm[5] := WSTRING#'PLC - el ajuste de barra de medición izquierda referencia no ok, manual de referencia (-8M1.L+SGV)';
   err[2174].alarm[6..8] := WSTRING#'';
   err[2175].alarm[1] := WSTRING#'PLC - Verstellung Messbalken links Referenzfahrt aktiv  (-8M1.L+SGV)';
   err[2175].alarm[2] := WSTRING#'PLC - adjustment metering bar left reference run active (-8M1.L+SGV)';
   err[2175].alarm[3] := WSTRING#'PLC - posizionamento barra di misura di sinistra corsa di riferimento attiva (-8M1.L+SGV)';
   err[2175].alarm[4] := WSTRING#'PLC - positionnement de barre de mesure gauche exécution de référence active (-8M1.L+SGV)';
   err[2175].alarm[5] := WSTRING#'PLC - el ajuste de barra de medición izquierda ejecución de referencia activa (-8M1.L+SGV)';
   err[2175].alarm[6..8] := WSTRING#'';
   err[2176].alarm[1] := WSTRING#'PLC - Verstellung Messbalken links nicht in Position (-8M1.L+SGV)';
   err[2176].alarm[2] := WSTRING#'PLC - adjustment metering bar left not in position (-8M1.L+SGV)';
   err[2176].alarm[3] := WSTRING#'PLC - posizionamento barra di misura di sinistra non in posizione (-8M1.L+SGV)';
   err[2176].alarm[4] := WSTRING#'PLC - positionnement de barre de mesure gauche pas en position (-8M1.L+SGV)';
   err[2176].alarm[5] := WSTRING#'PLC - el ajuste de barra de medición izquierda no está en posición (-8M1.L+SGV)';
   err[2176].alarm[6..8] := WSTRING#'';
   err[2177].alarm[1] := WSTRING#'PLC - Verstellung Messbalken links am Pc auf Hand geschalten (-8M1.L+SGV)';
   err[2177].alarm[2] := WSTRING#'PLC - adjustment metering bar left set on manual mode on Pc (-8M1.L+SGV)';
   err[2177].alarm[3] := WSTRING#'PLC - posizionamento barra di misura di sinistra attivata modalità manuale sul Pc (-8M1.L+SGV)';
   err[2177].alarm[4] := WSTRING#'PLC - positionnement de barre de mesure gauche passé en mode manuel sur le Pc (-8M1.L+SGV)';
   err[2177].alarm[5] := WSTRING#'PLC - el ajuste de barra de medición izquierda cambiado a manual en la Pc (-8M1.L+SGV)';
   err[2177].alarm[6..8] := WSTRING#'';
   err[2180].alarm[1] := WSTRING#'PLC - Störung Verstellung Messbalken rechts (-8M1.R+SGV)';
   err[2180].alarm[2] := WSTRING#'PLC - fault adjustment metering bar right (-8M1.R+SGV)';
   err[2180].alarm[3] := WSTRING#'PLC - errore posizionamento barra di misura di destra (-8M1.R+SGV)';
   err[2180].alarm[4] := WSTRING#'PLC - défaut positionnement de barre de mesure à droite (-8M1.R+SGV)';
   err[2180].alarm[5] := WSTRING#'PLC - fallo el ajuste de barra de medición derecha (-8M1.R+SGV)';
   err[2180].alarm[6..8] := WSTRING#'';
   err[2181].alarm[1] := WSTRING#'PLC - Störung Encoder - Verstellung Messbalken rechts (-8B1.R+SGV)';
   err[2181].alarm[2] := WSTRING#'PLC - fault encoder - adjustment metering bar right (-8B1.R+SGV)';
   err[2181].alarm[3] := WSTRING#'PLC - errore encoder - posizionamento barra di misura di destra (-8B1.R+SGV)';
   err[2181].alarm[4] := WSTRING#'PLC - défaut codeur - positionnement de barre de mesure à droite (-8B1.R+SGV)';
   err[2181].alarm[5] := WSTRING#'PLC - fallo codificador - el ajuste de barra de medición derecha (-8B1.R+SGV)';
   err[2181].alarm[6..8] := WSTRING#'';
   err[2182].alarm[1] := WSTRING#'PLC - Störung Sensor Endstellung links - Verstellung Messbalken rechts (-8S1.R+SGV)';
   err[2182].alarm[2] := WSTRING#'PLC - fault sensor limit switch position left - adjustment metering bar right (-8S1.R+SGV)';
   err[2182].alarm[3] := WSTRING#'PLC - errore sensore posizione sinistra - posizionamento barra di misura di destra (-8S1.R+SGV)';
   err[2182].alarm[4] := WSTRING#'PLC - défaut capteur position du fin de course à gauche - positionnement de barre de mesure à droite (-8S1.R+SGV)';
   err[2182].alarm[5] := WSTRING#'PLC - fallo sensor posición de límite a la izquierda - el ajuste de barra de medición derecha (-8S1.R+SGV)';
   err[2182].alarm[6..8] := WSTRING#'';
   err[2183].alarm[1] := WSTRING#'PLC - Störung Sensor Endstellung rechts - Verstellung Messbalken rechts (-8S2.R+SGV)';
   err[2183].alarm[2] := WSTRING#'PLC - fault sensor limit switch position right - adjustment metering bar right (-8S2.R+SGV)';
   err[2183].alarm[3] := WSTRING#'PLC - errore sensore posizione destra - posizionamento barra di misura di destra (-8S2.R+SGV)';
   err[2183].alarm[4] := WSTRING#'PLC - défaut capteur position du fin de course à droite - positionnement de barre de mesure à droite (-8S2.R+SGV)';
   err[2183].alarm[5] := WSTRING#'PLC - fallo sensor posición de límite a la derecha - el ajuste de barra de medición derecha (-8S2.R+SGV)';
   err[2183].alarm[6..8] := WSTRING#'';
   err[2184].alarm[1] := WSTRING#'PLC - Verstellung Messbalken rechts nicht referenziert, händisch neu referenzieren (-8M1.R+SGV)';
   err[2184].alarm[2] := WSTRING#'PLC - adjustment metering bar right reference not ok, reference manualy (-8M1.R+SGV)';
   err[2184].alarm[3] := WSTRING#'PLC - posizionamento barra di misura di destra riferimento non coretto, fare corsa di riferimento (-8M1.R+SGV)';
   err[2184].alarm[4] := WSTRING#'PLC - positionnement de barre de mesure à droite référence non correcte, manuel de référence (-8M1.R+SGV)';
   err[2184].alarm[5] := WSTRING#'PLC - el ajuste de barra de medición derecha referencia no ok, manual de referencia (-8M1.R+SGV)';
   err[2184].alarm[6..8] := WSTRING#'';
   err[2185].alarm[1] := WSTRING#'PLC - Verstellung Messbalken rechts Referenzfahrt aktiv  (-8M1.R+SGV)';
   err[2185].alarm[2] := WSTRING#'PLC - adjustment metering bar right reference run active (-8M1.R+SGV)';
   err[2185].alarm[3] := WSTRING#'PLC - posizionamento barra di misura di destra corsa di riferimento attiva (-8M1.R+SGV)';
   err[2185].alarm[4] := WSTRING#'PLC - positionnement de barre de mesure à droite exécution de référence active (-8M1.R+SGV)';
   err[2185].alarm[5] := WSTRING#'PLC - el ajuste de barra de medición derecha ejecución de referencia activa (-8M1.R+SGV)';
   err[2185].alarm[6..8] := WSTRING#'';
   err[2186].alarm[1] := WSTRING#'PLC - Verstellung Messbalken rechts nicht in Position (-8M1.R+SGV)';
   err[2186].alarm[2] := WSTRING#'PLC - adjustment metering bar right not in position (-8M1.R+SGV)';
   err[2186].alarm[3] := WSTRING#'PLC - posizionamento barra di misura di destra non in posizione (-8M1.R+SGV)';
   err[2186].alarm[4] := WSTRING#'PLC - positionnement de barre de mesure à droite pas en position (-8M1.R+SGV)';
   err[2186].alarm[5] := WSTRING#'PLC - el ajuste de barra de medición derecha no está en posición (-8M1.R+SGV)';
   err[2186].alarm[6..8] := WSTRING#'';
   err[2187].alarm[1] := WSTRING#'PLC - Verstellung Messbalken rechts am Pc auf Hand geschalten (-8M1.R+SGV)';
   err[2187].alarm[2] := WSTRING#'PLC - adjustment metering bar right set on manual mode on Pc (-8M1.R+SGV)';
   err[2187].alarm[3] := WSTRING#'PLC - posizionamento barra di misura di destra attivata modalità manuale sul Pc (-8M1.R+SGV)';
   err[2187].alarm[4] := WSTRING#'PLC - positionnement de barre de mesure à droite passé en mode manuel sur le Pc (-8M1.R+SGV)';
   err[2187].alarm[5] := WSTRING#'PLC - el ajuste de barra de medición derecha cambiado a manual en la Pc (-8M1.R+SGV)';
   err[2187].alarm[6..8] := WSTRING#'';
   err[2190].alarm[1] := WSTRING#'PLC - Störung Sensor für Distanzmessung von oben (-8B1+SGV)';
   err[2190].alarm[2] := WSTRING#'PLC - fault sensor distance measurement from top (-8B1+SGV)';
   err[2190].alarm[3] := WSTRING#'PLC - errore sensore misurazione della distanza dall`alto(-8B1+SGV)';
   err[2190].alarm[4] := WSTRING#'PLC - défaut capteur mesure de distance en haut (-8B1+SGV)';
   err[2190].alarm[5] := WSTRING#'PLC - fallo de sensor medición de distancia del sensor superior (-8B1+SGV)';
   err[2191].alarm[1] := WSTRING#'PLC - Störung Sensor für Distanzmessung von links (-8B2+SGV)';
   err[2191].alarm[2] := WSTRING#'PLC - fault sensor distance measurement from left (-8B2+SGV)';
   err[2191].alarm[3] := WSTRING#'PLC - errore sensore misurazione della distanza da sinistra (-8B2+SGV)';
   err[2191].alarm[4] := WSTRING#'PLC - défaut capteur mesure de distance de gauche à droite (-8B2+SGV)';
   err[2191].alarm[5] := WSTRING#'PLC - fallo de sensor medición de distancia del sensor desde la izquierda (-8B2+SGV)';
   err[2192].alarm[1] := WSTRING#'PLC - Störung Sensor für Distanzmessung von rechts (-8B3+SGV)';
   err[2192].alarm[2] := WSTRING#'PLC - fault sensor distance measurement from right (-8B3+SGV)';
   err[2192].alarm[3] := WSTRING#'PLC - errore sensore misurazione della distanza da destra (-8B3+SGV)';
   err[2192].alarm[4] := WSTRING#'PLC - défaut capteur mesure de distance de droite à gauche (-8B3+SGV)';
   err[2192].alarm[5] := WSTRING#'PLC - fallo de sensor medición de distancia del sensor desde la derecha (-8B3+SGV)';
   err[2200].alarm[1] := WSTRING#'PLC - Störung Profinet Slave LINMOT Servodrive - Verstellung Messbalken oben (-8U1.T+SGV)';
   err[2200].alarm[2] := WSTRING#'PLC - fault profinet-slave LINMOT Servodrive - adjustment metering bar top (-8U1.T+SGV)';
   err[2200].alarm[3] := WSTRING#'PLC - profinet-slave LINMOT Servodrive - posizionamento barra di misura superiore (-8U1.T+SGV)';
   err[2200].alarm[4] := WSTRING#'PLC - profinet-slave LINMOT Servodrive - positionnement de barre de mesure supérieure (-8U1.T+SGV)';
   err[2200].alarm[5] := WSTRING#'PLC - profinet-slave LINMOT Servodrive - el ajuste de barra de medición superior (-8U1.T+SGV)';
   err[2201].alarm[1] := WSTRING#'PLC - Störung Profinet Slave LINMOT Servodrive - Verstellung Messbalken links (-8U1.L+SGV)';
   err[2201].alarm[2] := WSTRING#'PLC - fault profinet-slave LINMOT Servodrive - adjustment metering bar left (-8U1.L+SGV)';
   err[2201].alarm[3] := WSTRING#'PLC - profinet-slave LINMOT Servodrive - posizionamento barra di misura di sinistra (-8U1.L+SGV)';
   err[2201].alarm[4] := WSTRING#'PLC - profinet-slave LINMOT Servodrive - positionnement de barre de mesure gauche (-8U1.L+SGV)';
   err[2201].alarm[5] := WSTRING#'PLC - profinet-slave LINMOT Servodrive - el ajuste de barra de medición izquierda (-8U1.L+SGV)';
   err[2202].alarm[1] := WSTRING#'PLC - Störung Profinet Slave LINMOT Servodrive - Verstellung Messbalken rechts (-8U1.R+SGV)';
   err[2202].alarm[2] := WSTRING#'PLC - fault profinet-slave LINMOT Servodrive - adjustment metering bar right (-8U1.R+SGV)';
   err[2202].alarm[3] := WSTRING#'PLC - profinet-slave LINMOT Servodrive - posizionamento barra di misura di destra(-8U1.R+SGV)';
   err[2202].alarm[4] := WSTRING#'PLC - profinet-slave LINMOT Servodrive - positionnement de barre de mesure à droite (-8U1.R+SGV)';
   err[2202].alarm[5] := WSTRING#'PLC - profinet-slave LINMOT Servodrive - el ajuste de barra de medición derecha (-8U1.R+SGV)';
END_DATA_BLOCK
